Staubli VAL3: SUB.dtx

public progItem pProg{}
